INTERFACE I_SimpleDynBuffer

PROPERTY Capacity : UDINT
GET
END_GET
END_PROPERTY

PROPERTY Empty : bool
GET
END_GET
END_PROPERTY

PROPERTY Full : bool
GET
END_GET
END_PROPERTY

METHOD Get : BOOL
VAR_INPUT
	pDestination : pvoid;
	cbSize : UDINT;
END_VAR
END_METHOD

METHOD Initialize : BOOL
VAR_INPUT
	nElementSize 		: UDINT;
	nElementCapacity 	: UDINT;
END_VAR
END_METHOD

METHOD Push : BOOL
VAR_INPUT
	pData : pvoid;
	cbSize : UDINT;
END_VAR
END_METHOD

METHOD Reset
END_METHOD

PROPERTY Size : UDINT
GET
END_GET
END_PROPERTY

END_INTERFACE

(* stored: Version 1.1.0.1
   Itf I_SimpleDynBuffer: Id {33a3ee71-0201-4e59-9750-de3c9f06ee75}
   Property Capacity: Id {acbfd4c0-7453-4bbd-8eb1-b9a410545ab1}
   Get Get: Id {6129ec76-23b0-4e5e-baef-80914c923d4d}
   Property Empty: Id {61a8b1d3-60ca-47dd-9fc2-43685a871626}
   Get Get: Id {ba3ebc72-19c4-4b46-9382-79d4dd9c35b4}
   Property Full: Id {0f98be4c-b59f-419e-acb1-112b6d08d1d5}
   Get Get: Id {943eb3ae-b093-485e-b952-a9479e1f51cf}
   Method Get: Id {2a2e9269-5fe0-49ef-9f44-88e9f07c1a07}
   Method Initialize: Id {94c7043f-ec22-4b52-94eb-e1a9671d92d7}
   Method Push: Id {11045d38-347b-4a4b-8864-172ae6cab984}
   Method Reset: Id {0ca36275-532e-4bed-8298-592b94af213e}
   Property Size: Id {b58b3b9c-78e3-4d9b-9969-331b9a853d2a}
   Get Get: Id {e3b936b4-5bed-45b5-9b75-bd3865e84fe1} *)
